{attribute 'qualified_only'}
VAR_GLOBAL CONSTANT
    bSkipDamperGripperForSimulation : BOOL := FALSE;
    bSkipAdjustGripperForSimulation : BOOL := FALSE;
END_VAR

(* stored: Version 1.1.0.1, ProductVersion 3.1.4026.20
   GVL GVL_SequenceConfig: Id {be476513-c5f5-46a2-b482-c989816bfc8f} *)
